Universal Robots PolyScope program: pittore_1.urp

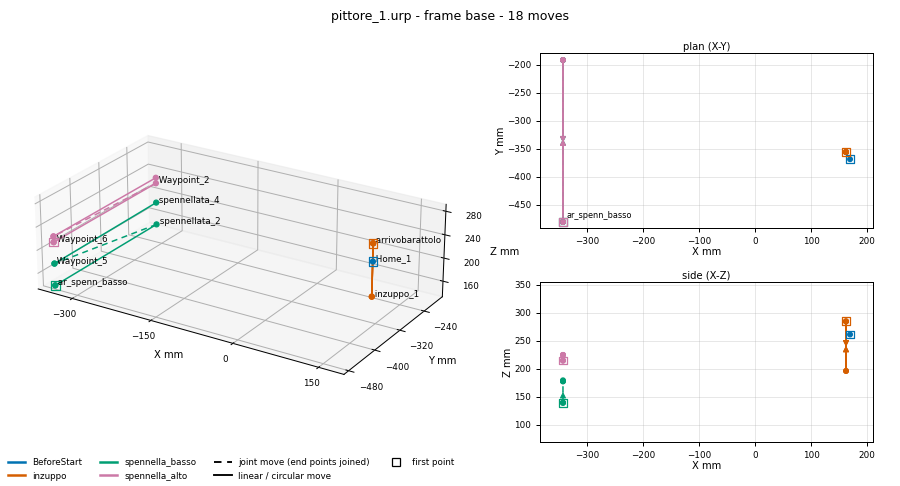
[picture p0: tool path of pittore_1.urp in frame base, 18 of 18 moves have a stored position in this frame; points joined in program order, loops and branches not executed]
Program pittore_1 (installation=default directory=/programs createdIn=3.15.8.106339 lastSavedIn=3.15.8.106339 robotSerialNumber=2021330429)
Calibrated DH parameters: a=[-0.000156, -0.236402, -0.171625, 0.000006, -0.000047, 0]; d=[0.151683, 29.702709, 78.973085, -108.563557, 0.085229, 0.082167]; alpha=[1.57015, 0.001987, 0.001164, 1.571718, -1.571778, 0]; deltaTheta=[-0.000066, 0.24449, 0.39032, -0.635025, 0.000068, -0.000043]
BeforeStart
  MoveJ speed 60 deg/s, acceleration 80 deg/s^2 (useActiveTCP=true)
    Waypoint Home_1: TCP in base x=169.233 y=-368.64 z=261.475 mm, rx=2.3406 ry=2.0166 rz=0.0586 rad; joints [309.389, -124.164, -13.951, -128.918, 92.336, 857.838] deg; flange x=159.446 y=-366.395 z=418.153 mm, rx=2.3406 ry=2.0166 rz=0.0586 rad
  URCap Gripper Activate (Robotiq_Grippers, Robotiq Inc.) dataModel(ResetAndActivateKey=false)
Robot Program (runOnlyOnce=false)
  Call inzuppo
  Call spennella_basso
  Call spennella_basso
  Call inzuppo
  Call spennella_alto
  Call spennella_alto
SubProgram -> spennella_alto
SubProgram -> spennella_basso
SubProgram -> inzuppo
SubProgram inzuppo (keepSynchronizedWithDisk=false)
  MoveJ speed 60 deg/s, acceleration 80 deg/s^2 (useActiveTCP=true)
    Waypoint arrivobarattolo: TCP in base x=162.033 y=-355.947 z=284.852 mm, rx=2.2788 ry=2.023 rz=-0.0015 rad; joints [311.206, -117.832, -18.362, -128.327, 90.07, 857.894] deg; flange x=152.317 y=-344.777 z=441.152 mm, rx=2.2788 ry=2.023 rz=-0.0015 rad
    MoveL speed 250 mm/s, acceleration 1200 mm/s^2 (useActiveTCP=true) feature=Base
      Waypoint inzuppo_1: TCP in base x=162.074 y=-355.899 z=196.398 mm, rx=2.2788 ry=2.0233 rz=-0.0013 rad; joints [311.249, -103.715, -66.047, -94.772, 90.077, 857.943] deg; flange x=152.371 y=-344.766 z=352.702 mm, rx=2.2788 ry=2.0233 rz=-0.0013 rad
      Waypoint esco_inzuppo_1: TCP in base x=162.006 y=-355.943 z=284.851 mm, rx=2.2788 ry=2.023 rz=-0.0015 rad; joints [311.205, -117.831, -18.362, -128.331, 90.068, 857.893] deg; flange x=152.3 y=-344.775 z=441.152 mm, rx=2.2788 ry=2.023 rz=-0.0015 rad
      Waypoint inzuppo_2: TCP in base x=162.095 y=-355.912 z=196.394 mm, rx=2.2787 ry=2.0233 rz=-0.0014 rad; joints [311.254, -103.717, -66.047, -94.769, 90.073, 857.945] deg; flange x=152.398 y=-344.768 z=352.697 mm, rx=2.2787 ry=2.0233 rz=-0.0014 rad
      Waypoint esco_inzuppo_2: TCP in base x=162.01 y=-355.969 z=284.833 mm, rx=2.2789 ry=2.0229 rz=-0.0015 rad; joints [311.203, -117.838, -18.357, -128.33, 90.068, 857.896] deg; flange x=152.306 y=-344.802 z=441.134 mm, rx=2.2789 ry=2.0229 rz=-0.0015 rad
SubProgram spennella_basso (keepSynchronizedWithDisk=false)
  MoveJ speed 60 deg/s, acceleration 80 deg/s^2 (useActiveTCP=true)
    Waypoint ar_spenn_basso: TCP in base x=-342.979 y=-480.431 z=139.764 mm, rx=-1.339 ry=-1.1513 rz=1.3241 rad; joints [271.086, -149.634, -60.943, -74.382, 1.403, 834.228] deg; flange x=-186.021 y=-478.707 z=142.981 mm, rx=-1.339 ry=-1.1513 rz=1.3241 rad
    MoveL speed 250 mm/s, acceleration 1200 mm/s^2 (useActiveTCP=true) feature=Base
      Waypoint spennellata_1: TCP in base x=-342.984 y=-480.419 z=139.742 mm, rx=-1.3391 ry=-1.1513 rz=1.3241 rad; joints [271.085, -149.634, -60.945, -74.377, 1.408, 834.226] deg; flange x=-186.027 y=-478.7 z=142.972 mm, rx=-1.3391 ry=-1.1513 rz=1.3241 rad
      Waypoint spennellata_2: TCP in base x=-342.984 y=-191.635 z=139.689 mm, rx=-1.3391 ry=-1.1513 rz=1.324 rad; joints [272.68, -95.006, -141.763, -90.342, 2.332, 876.398] deg; flange x=-186.027 y=-189.929 z=142.931 mm, rx=-1.3391 ry=-1.1513 rz=1.324 rad
      MoveJ speed 60 deg/s, acceleration 80 deg/s^2 (useActiveTCP=true)
        Waypoint Waypoint_5: TCP in base x=-343 y=-480.41 z=177.906 mm, rx=-1.339 ry=-1.1513 rz=1.324 rad; joints [271.082, -144.912, -59.428, -80.128, 1.397, 833.733] deg; flange x=-186.043 y=-478.699 z=181.135 mm, rx=-1.339 ry=-1.1513 rz=1.324 rad
      Waypoint spennellata_3: TCP in base x=-342.995 y=-480.412 z=177.901 mm, rx=-1.339 ry=-1.1513 rz=1.3241 rad; joints [271.083, -144.912, -59.432, -80.124, 1.393, 833.736] deg; flange x=-186.037 y=-478.696 z=181.121 mm, rx=-1.339 ry=-1.1513 rz=1.3241 rad
      Waypoint spennellata_4: TCP in base x=-342.987 y=-191.611 z=179.749 mm, rx=-1.3391 ry=-1.1513 rz=1.3239 rad; joints [272.68, -84.267, -135.995, -107.047, 2.313, 876.593] deg; flange x=-186.03 y=-189.909 z=182.989 mm, rx=-1.3391 ry=-1.1513 rz=1.3239 rad
SubProgram spennella_alto (keepSynchronizedWithDisk=false)
  MoveJ speed 60 deg/s, acceleration 80 deg/s^2 (useActiveTCP=true)
    Waypoint Waypoint_6: TCP in base x=-342.983 y=-480.418 z=215.044 mm, rx=-1.3387 ry=-1.1513 rz=1.3241 rad; joints [271.082, -141.26, -56.169, -86.571, 1.372, 833.259] deg; flange x=-186.025 y=-478.693 z=218.236 mm, rx=-1.3387 ry=-1.1513 rz=1.3241 rad
    MoveL speed 250 mm/s, acceleration 1200 mm/s^2 (useActiveTCP=true) feature=Base
      Waypoint Waypoint_1: TCP in base x=-343 y=-480.394 z=215.03 mm, rx=-1.3389 ry=-1.1513 rz=1.3239 rad; joints [271.08, -141.257, -56.164, -86.58, 1.384, 833.263] deg; flange x=-186.042 y=-478.683 z=218.253 mm, rx=-1.3389 ry=-1.1513 rz=1.3239 rad
      Waypoint Waypoint_2: TCP in base x=-342.997 y=-191.6 z=215.015 mm, rx=-1.3392 ry=-1.1512 rz=1.3239 rad; joints [272.68, -78.012, -129.432, -120.046, 2.3, 876.779] deg; flange x=-186.04 y=-189.908 z=218.253 mm, rx=-1.3392 ry=-1.1512 rz=1.3239 rad
      MoveJ speed 60 deg/s, acceleration 80 deg/s^2 (useActiveTCP=true)
        Waypoint Waypoint_7: TCP in base x=-342.976 y=-480.408 z=225.039 mm, rx=-1.3389 ry=-1.1514 rz=1.3239 rad; joints [271.082, -140.454, -54.954, -88.464, 1.383, 833.133] deg; flange x=-186.019 y=-478.691 z=228.268 mm, rx=-1.3389 ry=-1.1514 rz=1.3239 rad
      Waypoint Waypoint_3: TCP in base x=-342.982 y=-480.405 z=225.044 mm, rx=-1.3389 ry=-1.1513 rz=1.324 rad; joints [271.081, -140.454, -54.955, -88.462, 1.382, 833.132] deg; flange x=-186.024 y=-478.69 z=228.269 mm, rx=-1.3389 ry=-1.1513 rz=1.324 rad
      Waypoint Waypoint_4: TCP in base x=-342.986 y=-191.616 z=225.013 mm, rx=-1.3391 ry=-1.1513 rz=1.3239 rad; joints [272.684, -76.718, -127.368, -123.458, 2.297, 876.829] deg; flange x=-186.028 y=-189.913 z=228.249 mm, rx=-1.3391 ry=-1.1513 rz=1.3239 rad
